FUNCTION TryConvert_REAL_TO_WORD : BOOL
VAR_INPUT
	in : REAL;
	out : REFERENCE TO WORD;
END_VAR

IF in > DatatypeLimits.MAX_VALUE_OF_REAL_WHICH_CAN_BE_HELD_IN_A_WORD THEN
	RETURN;
END_IF

IF in < DatatypeLimits.MIN_VALUE_OF_REAL_WHICH_CAN_BE_HELD_IN_A_WORD THEN
	RETURN;
END_IF

out := REAL_TO_WORD(in);
TryConvert_REAL_TO_WORD := TRUE;

END_FUNCTION

(* stored: Version 1.1.0.1, ProductVersion 3.1.4024.12
   POU TryConvert_REAL_TO_WORD: Id {3ffd57bf-3cd0-404f-850f-80f45923b199}, SpecialFunc None *)
